{attribute 'TcGenerated'}
// This function has been automatically generated from the project information.
VAR_GLOBAL CONSTANT
	{attribute 'const_non_replaced'}
	{attribute 'linkalways'}
	stLibVersion_lcls_twincat_motion_sheppard : ST_LibVersion := (iMajor := 0, iMinor := 0, iBuild := 0, iRevision := 0, sVersion := '0.0.0');
END_VAR

(* stored: Version 1.1.0.1, ProductVersion 3.1.4020.14
   GVL Global_Version: Id {31efc82a-653f-4c8c-bd59-d2d2aaf902fa} *)
